TYPE ST_Vise_Status :
STRUCT
	eState			:E_Vise_State;		//
	eSocketState	:E_ViseSocketState;
	bPass			:BOOL;
	bFail			:BOOL;
	nViseIndex		:USINT; // 1-14
END_STRUCT
END_TYPE

(* stored: Version 1.1.0.1, ProductVersion 3.1.4024.12
   DUT ST_Vise_Status: Id {ae77624c-a36f-44e8-9619-c4fb608f31d3} *)
